{attribute 'qualified_only'}
{attribute 'strict'}
TYPE GCControllerMode :
(
	CurrentControlled,
	ForceControlled
);
END_TYPE

(* stored: Version 1.1.0.1, ProductVersion 3.1.4024.12
   DUT GCControllerMode: Id {46af96ec-5c12-4b2a-be60-8306c3b7817f} *)
